ABB RobotStudio station: Eksamens_færdigt_udkast_14-05_16.24.rspag

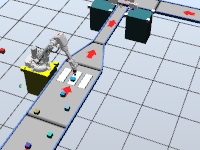
--- station ---
Station Eksamens (saved by RobotStudio 7.0.8746.631)
Controller Virtual_controller, task T_ROB3: task frame (RAPID world) sits at (-5805.06, 703.5, 890) mm, rotated rx 0 ry 0 rz -90 deg in the station
Controller Virtual_controller, task T_ROB2: task frame (RAPID world) sits at (-5805.06, 703.5, 890) mm, rotated rx 0 ry 0 rz -90 deg in the station
Controller Virtual_controller, task T_ROB1: task frame (RAPID world) sits at (-5805.06, 703.5, 890) mm, rotated rx 0 ry 0 rz -90 deg in the station
Controller Virtual_controller
  mechanical unit ROB_1: IRB120_3_58__01_2, 6 joints, base frame (83.5, -144.94, 0) mm
  mechanical unit ROB_2: IRB2600_20_165_C_01_2, 6 joints, base frame (1331.39, 3332.7, 0) mm, rotated rx 0 ry 0 rz 180 deg
  mechanical unit ROB_3: IRB120_3_58__01_3, 6 joints, base frame (643.5, -144.94, 0) mm, rotated rx 0 ry 0 rz 180 deg
Layout (positions relative to the parent item):
  - Sorter_kasser [graphiccomponentgroup]
    - Assemblies [graphiccomponentgroup]
      - Section1 [graphiccomponentgroup]
        - ABB_IRC5_ctrl [graphiccomponentgroup]
          - ABB_IRC5_ctrl_1 [graphiccomponentgroup]
            - Mesh0 [part]
        - Conveyor__Straight_ [graphiccomponentgroup]
          - CONVEYOR1 [graphiccomponentgroup]
            - Mesh1 [part]
            - Mesh2 [part]
            - Mesh3 [part]
          - CONVEYOR2 [graphiccomponentgroup]
            - Mesh4 [part]
            - Mesh5 [part]
            - Mesh6 [part]
          - CONVEYOR3 [graphiccomponentgroup]
            - Mesh7 [part]
            - Mesh8 [part]
            - Mesh9 [part]
          - CONVEYOR4 [graphiccomponentgroup]
            - Mesh10 [part]
            - Mesh11 [part]
            - Mesh12 [part]
          - CONVEYOR5 [graphiccomponentgroup]
            - Mesh13 [part]
            - Mesh14 [part]
            - Mesh15 [part]
          - CONVEYOR6 [graphiccomponentgroup]
            - Mesh16 [part]
            - Mesh17 [part]
            - Mesh18 [part]
          - CONVEYOR7 [graphiccomponentgroup]
            - Mesh19 [part]
            - Mesh20 [part]
            - Mesh21 [part]
        - Cube [graphiccomponentgroup]
          - Cube1 [graphiccomponentgroup]
            - Mesh22 [part]
            - Mesh23 [part]
            - Mesh24 [part]
            - Mesh25 [part]
            - Mesh26 [part]
          - Cube2 [graphiccomponentgroup]
            - Mesh27 [part]
            - Mesh28 [part]
            - Mesh29 [part]
            - Mesh30 [part]
            - Mesh31 [part]
          - Cube3 [graphiccomponentgroup]
            - Mesh32 [part]
            - Mesh33 [part]
            - Mesh34 [part]
            - Mesh35 [part]
            - Mesh36 [part]
        - Eater [graphiccomponentgroup]
          - EATER1 [graphiccomponentgroup]
            - Mesh37 [part]
        - Display [graphiccomponentgroup]
          - EaterSmall [graphiccomponentgroup]
            - Mesh38 [part]
            - Mesh39 [part]
            - Mesh40 [part]
            - Mesh41 [part]
            - Mesh42 [part]
            - Mesh43 [part]
            - Mesh44 [part]
            - Mesh45 [part]
            - Mesh46 [part]
            - Mesh47 [part]
            - Mesh48 [part]
        - Feeder [graphiccomponentgroup]
          - FEEDER1 [graphiccomponentgroup]
            - Mesh49 [part]
            - Mesh50 [part]
          - FEEDER2 [graphiccomponentgroup]
            - Mesh51 [part]
            - Mesh52 [part]
          - FEEDER3 [graphiccomponentgroup]
            - Mesh53 [part]
            - Mesh54 [part]
        - Scale [graphiccomponentgroup]
          - Scale_Weight [graphiccomponentgroup]
            - Mesh55 [part]
            - Mesh56 [part]
            - Mesh57 [part]
            - Mesh58 [part]
          - Scale_Weight1 [graphiccomponentgroup]
            - Mesh59 [part]
            - Mesh60 [part]
            - Mesh61 [part]
            - Mesh62 [part]
          - Scale_Weight2 [graphiccomponentgroup]
            - Mesh63 [part]
            - Mesh64 [part]
            - Mesh65 [part]
            - Mesh66 [part]
        - Text [graphiccomponentgroup]
          - Text1 [graphiccomponentgroup]
            - Mesh67 [part]
    - Motors [graphiccomponentgroup]
      - Surface [graphiccomponentgroup]
        - MOTOR1 [graphiccomponentgroup]
          - Mesh75 [part]
          - Mesh76 [part]
          - Mesh77 [part]
          - Mesh78 [part]
        - MOTOR6 [graphiccomponentgroup]
          - Mesh79 [part]
        - MOTOR8 [graphiccomponentgroup]
          - Mesh80 [part]
        - MOTOR9 [graphiccomponentgroup]
          - Mesh81 [part]
    - Loads [graphiccomponentgroup]
      - Mesh68 [part]
      - Mesh69 [part]
      - Mesh70 [part]
      - Mesh71 [part]
      - Mesh72 [part]
      - Mesh73 [part]
      - Mesh74 [part]
  - IRB120_3_58__01_2 [mechanism, from Robots\IRB120_3_58_G_01.rslib] at (-5950, 620, 890) mm, rotated rx 0 ry 0 rz -90 deg; joint values [-0.0063, -0.4744, 1.1199, 0, 0.9253, -0.0063] (rad or m)
  - IRB2600_20_165_C_01_2 [mechanism, from Robots\IRB2600_20_165_C_01.rslib] at (-2472.36, -627.89, 890) mm, rotated rx 0 ry 0 rz 90 deg; joint values [-0.0004, 0.5644, 0.5607, 0, 0.4457, -0.0004] (rad or m)
  - IRB120_3_58__01_3 [mechanism, from Robots\IRB120_3_58_G_01.rslib] at (-5950, 60, 890) mm, rotated rx 0 ry 0 rz 90 deg; joint values [0.006, -0.4425, 1.1015, 0, 0.9118, 0.006] (rad or m)
  - GripperStackerRight [mechanism] at (-5951, 460, 1222.41) mm, rotated rx 180 ry 0 rz 90 deg
      TCP GripperStackerRight at (0, 0, 30) mm
      links: SimpleGripper
  - GripperStackerLeft [mechanism] at (-5951, 226, 1222.41) mm, rotated rx -180 ry 0 rz -90 deg
      TCP GripperStackerLeft at (0, 0, 30) mm
      links: SimpleGripper
  - GripperSorter [mechanism] at (-2472, 343, 1173.67) mm, rotated rx -180 ry 0 rz -90 deg
      TCP GripperSorter at (0, 0, 30) mm
      links: SimpleGripper
Attachment: GripperStackerRight is attached to IRB120_3_58__01_2 / Link6
Attachment: GripperStackerLeft is attached to IRB120_3_58__01_3 / Link6
Attachment: GripperSorter is attached to IRB2600_20_165_C_01_2 / Link6

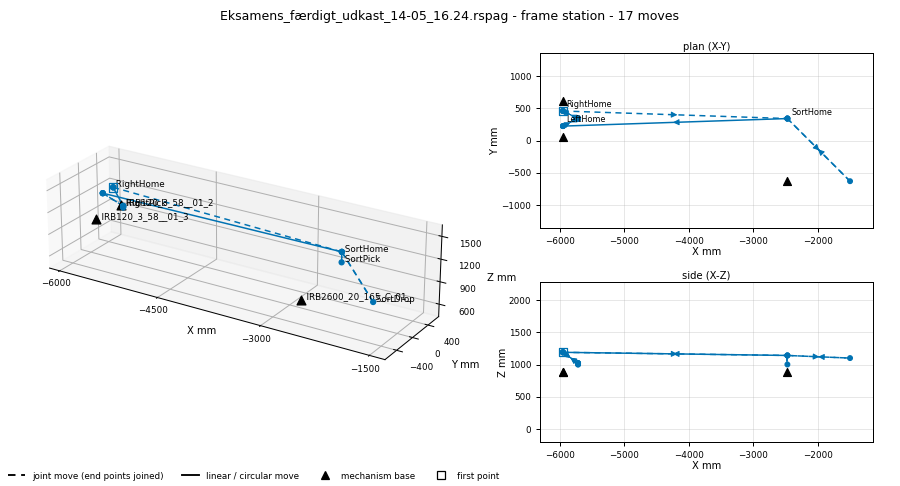
[picture p0: tool path of Eksamens_færdigt_udkast_14-05_16.24.rspag in frame station, 17 of 19 moves have a stored position in this frame; points joined in program order, loops and branches not executed]
--- Backups/Virtual_controller/RAPID/TASK1/PROGMOD/CalibData.mod ---
MODULE CalibData
	PERS tooldata GripperStackerRight:=[TRUE,[[0,0,30],[1,0,0,0]],[1,[0,0,1],[1,0,0,0],0,0,0]];
ENDMODULE

--- Backups/Virtual_controller/RAPID/TASK1/PROGMOD/Module1.mod ---
MODULE Module1
    CONST robtarget RightPick:=[[360.5,88.055,133.879],[0,0,1,0],[0,0,0,0],[9E+09,9E+09,9E+09,9E+09,9E+09,9E+09]];
    CONST robtarget Right11:=[[305.5,-515.945,197.406],[0,0,1,0],[-1,0,-1,0],[9E+09,9E+09,9E+09,9E+09,9E+09,9E+09]];
    CONST robtarget Right12:=[[305.5,-625.945,197.406],[0,0,1,0],[-1,0,-1,0],[9E+09,9E+09,9E+09,9E+09,9E+09,9E+09]];
    CONST robtarget Right21:=[[305.5,-515.945,302.406],[0,0,1,0],[-1,0,-1,0],[9E+09,9E+09,9E+09,9E+09,9E+09,9E+09]];
    CONST robtarget Right22:=[[305.5,-625.945,302.406],[0,0,1,0],[-1,0,-1,0],[9E+09,9E+09,9E+09,9E+09,9E+09,9E+09]];
    CONST robtarget RightHome:=[[243.5,-145.945,302.406],[0,0,1,0],[-1,0,-1,0],[9E+09,9E+09,9E+09,9E+09,9E+09,9E+09]];

    ! Init data
    VAR num stackCount := 0;
    VAR robtarget tempTarget;
    VAR speeddata speed := v7000;
    VAR bool init := TRUE;
    !***********************************************************
    !
    ! Module:  Right Stacker robot
    !
    ! Description:
    !   <Insert description here>
    !
    ! Author: madsw
    ! Version: 1.0
    !
    !***********************************************************
    PROC main()
        ! Checking if all do's are correctly reset.
        IF init THEN
            init := FALSE;
            initProc;
            MoveL RightHome, speed, z100, GripperStackerRight;
            WaitRob \InPos;
        ENDIF

            ! Move when There is and object and Left arm is not in the way.
        IF (diStackerRightPick = 1 OR diStackerPick = 1) AND
           ((NOT doStackDone = 1) OR (NOT doStackerRightDone = 1)) THEN

                ! picking up, Claiming Pickup token if available.
            IF doStackerLeftPickingUp = 0 AND LeftWentLast = 1 THEN
                    ! Moving in to pick up while claiming Pickup token.
                SetDO doStackerRightPickingUp, 1;
                WaitDO doStackerRightPickingUp, 1;
                SetDO LeftWentLast, 0;
                WaitDO LeftWentLast, 0;

                    ! Grippping with wait.
                SetDO doStackerRightGripper, 1;
                WaitDO doStackerRightGripper, 1;
                MoveJ RightPick, speed, z100, GripperStackerRight;
                MoveJ Offs(RightPick, 0, 0, -20), speed, z100, GripperStackerRight;
                WaitRob \InPos;

                WaitTime(0.2);
                    ! Moving out, unclaiming pickup token.
                MoveJ RightPick, speed, z100, GripperStackerRight;
                MoveJ RightHome, speed, z100, GripperStackerRight;
                WaitRob \InPos;

                SetDO doStackerRightDelivering, 1;
                WaitDO doStackerRightDelivering, 1;
                SetDO doStackerRightPickingUp, 0;
                WaitDO doStackerRightPickingUp, 0;

                    ! Pickup token unclaimed, and moving in to place block.
                stackCount := stackCount +1;
                TEST stackCount
                CASE 1:
                    tempTarget := Right12;
                CASE 2:
                    tempTarget := Right11;
                CASE 3:
                    tempTarget := Right22;
                CASE 4:
                    tempTarget := Right21;
                DEFAULT:
                    TPWrite "Something went wrong.";
                ENDTEST

                MoveL tempTarget, speed, z100, GripperStackerRight;
                WaitRob \InPos;

                SetDO doStackerRightGripper, 0;
                WaitDO doStackerRightGripper, 0;
                WaitTime(0.3);

                ! Moving home
                MoveL RightHome, speed, z100, GripperStackerRight;
                WaitRob \InPos;
                SetDO doStackerRightDelivering, 0;
                WaitDO doStackerRightDelivering, 0;
            ENDIF
        ENDIF

        ! If the resetStackers signal is recieved we reset
        IF diResetStackers = 1 THEN
            stackCount := 0;
            SetDO doStackerRightDone, 0;
            WaitDO doStackerRightDone, 0;
            IF doStackerLeftDone = 0 AND doStackDone = 1 THEN
                SetDO doStackDone, 0;
                WaitDO doStackDone, 0;
            ENDIF
        ENDIF

        ! If the stackcount has reached 4 this side of the stack is done.
        IF stackCount = 4 THEN
            SetDO doStackerRightDone, 1;
            WaitDO doStackerRightDone, 1;
            IF doStackerLeftDone = 1 THEN
                SetDO doStackDone, 1;
                WaitDO doStackDone, 1;
            ENDIF
        ENDIF
    ENDPROC

    ! Init program
    PROC initProc()
        SetDO doStackerRightDelivering, 0;
        SetDO doStackerRightGripper, 0;
        SetDO doStackerRightPickingUp, 0;
        SetDO doStackerLeftDone, 0;
        SetDO doStackDone, 0;
        WaitDO doStackerLeftDone, 0;
        WaitDO doStackDone, 0;
        WaitDO doStackerRightDelivering, 0;
        WaitDO doStackerRightGripper, 0;
        WaitDO doStackerRightPickingUp, 0;
    ENDPROC
ENDMODULE

--- Backups/Virtual_controller/RAPID/TASK2/PROGMOD/CalibData.mod ---
MODULE CalibData
	PERS tooldata GripperSorter:=[TRUE,[[0,0,30],[1,0,0,0]],[1,[0,0,1],[1,0,0,0],0,0,0]];
ENDMODULE

--- Backups/Virtual_controller/RAPID/TASK2/PROGMOD/Module1.mod ---
MODULE Module1
    CONST robtarget SortPick:=[[360.5,3333.055,113.666],[0,1,0,0],[-1,0,-1,0],[9E+09,9E+09,9E+09,9E+09,9E+09,9E+09]];
    CONST robtarget SortDrop:=[[1331.5,4304.055,212.998],[0,-0.707106781,0.707106781,0],[-2,0,-1,0],[9E+09,9E+09,9E+09,9E+09,9E+09,9E+09]];
    CONST robtarget SortHome:=[[360.5,3333.055,253.666],[0,1,0,0],[-1,0,-1,0],[9E+09,9E+09,9E+09,9E+09,9E+09,9E+09]];

    VAR speeddata speed := v7000;
    VAR bool init := TRUE;
    !***********************************************************
    !
    ! Module:  Sorter robot
    !
    ! Description:
    !   <Insert description here>
    !
    ! Author: madsw
    ! Version: 1.0
    !
    !***********************************************************

    PROC main()
        IF init THEN
            init := FALSE;
            initProc;
            MoveJ SortHome, speed, z100, GripperSorter;
            WaitRob \inpos;
        ENDIF

        IF diSorterPick = 1 THEN
                ! Move to grip.
            SetDO doSorterGripper, 1;
            WaitDO doSorterGripper, 1;
            MoveJ SortPick, speed, z100, GripperSorter;
            WaitRob \InPos;

            WaitTime(0.2);
            SetDO doSorterDelivering, 1;
            WaitDO doSorterDelivering, 1;
                ! Move to drop.
            MoveJ SortHome, speed, z100, GripperSorter;
            MoveJ SortDrop, speed, z100, GripperSorter;
            WaitRob \InPos;
            SetDO doSorterGripper, 0;
            WaitDO doSorterGripper, 0;
            WaitTime(0.3);

            ! Moving home and resetting
            MoveJ SortHome, speed, z100, GripperSorter;
            WaitRob \inpos;
            SetDO doSorterDelivering, 0;
            WaitDO doSorterDelivering, 0;
        ENDIF
    ENDPROC

    ! Init program
    PROC initProc()
        SetDO doSorterGripper, 0;
        SetDO doSorterDelivering, 0;
        WaitDO doSorterDelivering, 0;
        WaitDO doSorterGripper, 0;
    ENDPROC
ENDMODULE

--- Backups/Virtual_controller/RAPID/TASK3/PROGMOD/CalibData.mod ---
MODULE CalibData
    PERS tooldata GripperStackerLeft:=[TRUE,[[0,0,30],[1,0,0,0]],[1,[0,0,1],[1,0,0,0],0,0,0]];
ENDMODULE

--- Backups/Virtual_controller/RAPID/TASK3/PROGMOD/Module1.mod ---
MODULE Module1
    CONST robtarget LeftPick:=[[360.5,88.055,133.879],[0,1,0,0],[-1,0,-1,0],[9E+09,9E+09,9E+09,9E+09,9E+09,9E+09]];
    CONST robtarget Left11:=[[415.5,-515.945,197.406],[0,1,0,0],[0,0,0,0],[9E+09,9E+09,9E+09,9E+09,9E+09,9E+09]];
    CONST robtarget Left12:=[[415.5,-625.945,197.406],[0,1,0,0],[0,0,0,0],[9E+09,9E+09,9E+09,9E+09,9E+09,9E+09]];
    CONST robtarget Left21:=[[415.5,-515.945,302.406],[0,1,0,0],[0,0,0,0],[9E+09,9E+09,9E+09,9E+09,9E+09,9E+09]];
    CONST robtarget Left22:=[[415.5,-625.945,302.406],[0,1,0,0],[0,0,0,0],[9E+09,9E+09,9E+09,9E+09,9E+09,9E+09]];
    CONST robtarget LeftHome:=[[477.5,-145.945,302.406],[0,1,0,0],[0,0,0,0],[9E+09,9E+09,9E+09,9E+09,9E+09,9E+09]];

    VAR num stackCount := 0;
    VAR robtarget tempTarget;
    VAR speeddata speed := v7000;
    VAR bool init := TRUE;
    !***********************************************************
    !
    ! Module:  Left Stacker robot
    !
    ! Description:
    !   <Insert description here>
    !
    ! Author: madsw
    ! Version: 1.0
    !
    !***********************************************************
    PROC main()
        ! Checking if all do's are correctly reset.
        IF init THEN
            init := FALSE;
            initProc;
            MoveL LeftHome, speed, z100, GripperStackerLeft;
            WaitRob \InPos;
        ENDIF

            ! Move when There is and object and Left arm is not in the way.
        IF diStackerLeftPick = 1 OR diStackerPick = 1  AND
           ((NOT doStackDone = 1) OR (NOT doStackerLeftDone = 1)) THEN

                ! picking up, Claiming Pickup token if available.
            IF (doStackerRightPickingUp = 0 AND LeftWentLast = 0) THEN
                    ! Moving in to pick up while claiming Pickup token.
                SetDO doStackerLeftPickingUp, 1;
                WaitDO doStackerLeftPickingUp, 1;
                SetDO LeftWentLast, 1;
                WaitDO LeftWentLast, 1;

                    ! Grippping with wait.
                SetDO doStackerLeftGripper, 1;
                WaitDO doStackerLeftGripper, 1;
                MoveJ LeftPick, speed, z100, GripperStackerLeft;
                MoveJ Offs(LeftPick, 0, 0, -20), speed, z100, GripperStackerLeft;
                WaitRob \InPos;

                WaitTime(0.2);
                    ! Moving out, unclaiming pickup token.
                MoveJ LeftPick, speed, z100, GripperStackerLeft;
                MoveJ LeftHome, speed, z100, GripperStackerLeft;
                WaitRob \InPos;

                SetDO doStackerLeftDelivering, 1;
                WaitDO doStackerLeftDelivering, 1;
                SetDO doStackerLeftPickingUp, 0;
                WaitDO doStackerLeftPickingUp, 0;

                    ! Pickup token unclaimed, and moving in to place block.
                stackCount := stackCount +1;
                TEST stackCount
                CASE 1:
                    tempTarget := Left12;
                CASE 2:
                    tempTarget := Left11;
                CASE 3:
                    tempTarget := Left22;
                CASE 4:
                    tempTarget := Left21;
                DEFAULT:
                    TPWrite "Something went wrong";
                ENDTEST

                MoveL tempTarget, speed, z100, GripperStackerLeft;
                WaitRob \InPos;

                SetDO doStackerLeftGripper, 0;
                WaitDO doStackerLeftGripper, 0;
                WaitTime(0.3);

                ! Moving home
                MoveL LeftHome, speed, z100, GripperStackerLeft;
                WaitRob \InPos;
                SetDO doStackerLeftDelivering, 0;
                WaitDO doStackerLeftDelivering, 0;
            ENDIF
        ENDIF

        ! If the resetStackers signal is recieved we reset
        IF diResetStackers = 1 THEN
            stackCount := 0;
            SetDO doStackerLeftDone, 0;
            WaitDO doStackerLeftDone, 0;
            IF doStackerRightDone = 0 AND doStackDone = 1 THEN
                SetDO doStackDone, 0;
                WaitDO doStackDone, 0;
            ENDIF
        ENDIF

        ! If the stackcount has reached 4 this side of the stack is done.
        IF stackCount = 4 THEN
            SetDO doStackerLeftDone, 1;
            WaitDO doStackerLeftDone, 1;
            IF doStackerRightDone = 1 THEN
                SetDO doStackDone, 1;
                WaitDO doStackDone, 1;
            ENDIF
        ENDIF
    ENDPROC

    ! Init program
    PROC initProc()
        SetDO doStackerLeftDelivering, 0;
        SetDO doStackerLeftGripper, 0;
        SetDO doStackerLeftPickingUp, 0;
        SetDO doStackerLeftDone, 0;
        SetDO doStackDone, 0;
        WaitDO doStackerLeftDone, 0;
        WaitDO doStackDone, 0;
        WaitDO doStackerLeftDelivering, 0;
        WaitDO doStackerLeftGripper, 0;
        WaitDO doStackerLeftPickingUp, 0;
    ENDPROC
ENDMODULE

--- Backups/Virtual_controller/SYSPAR/EIO.cfg ---
EIO:CFG_1.0:6:1::
#
EIO_SIGNAL:

      -Name "diSorterPick" -SignalType "DI" -Access "All"

      -Name "diStackerRightPick" -SignalType "DI" -Access "All"

      -Name "diStackerLeftPick" -SignalType "DI" -Access "All"

      -Name "doStackerRightGripper" -SignalType "DO" -Access "All"

      -Name "doStackerLeftGripper" -SignalType "DO" -Access "All"

      -Name "doSorterGripper" -SignalType "DO" -Access "All"

      -Name "doStackerRightPickingUp" -SignalType "DO" -Access "All"

      -Name "doStackerLeftPickingUp" -SignalType "DO" -Access "All"

      -Name "doStackerRightDelivering" -SignalType "DO" -Access "All"

      -Name "doStackerLeftDelivering" -SignalType "DO" -Access "All"

      -Name "doStackerRightDone" -SignalType "DO" -Access "All"

      -Name "doStackerLeftDone" -SignalType "DO" -Access "All"

      -Name "LeftWentLast" -SignalType "DO" -Access "All"

      -Name "diStackerPick" -SignalType "DI" -Access "All"

      -Name "doStackDone" -SignalType "DO" -Access "All"

      -Name "doSorterDelivering" -SignalType "DO" -Access "All"

      -Name "diResetStackers" -SignalType "DI" -Access "All"
